(* Logix 5000 project; controller CHASKEY Emulate 5570 rev 30.12; software revision 30.00 *)

TASK MainTask (periodic, rate 3000 ms, priority 1, watchdog 5000 ms) : MainProgram

MODULES
   Local : Emulate 5570 (ICP 2, rev 30.12)
END_MODULES

VAR_GLOBAL   (* controller tags *)
   _SEC_P : BOOL;
   done : DINT;
   R_TRIG : FBD_ONESHOT;
   temp_var : DINT;
   test_array : DINT[20] := ([0] := 1, [1] := 2, [2] := 3, [3] := 4, [4] := 5, [5] := 6, [6] := 7, [7] := 8, [8] := 9, [9] := 10, [10] := 11, [11] := 12, [12] := 13, [13] := 14, [14] := 15, [15] := 16, [16] := 17, [17] := 18, [18] := 19, [19] := 20);
   TON : FBD_TIMER;
END_VAR

PROGRAM MainProgram   (* main routine MainRoutine *)
VAR
   Chaskey_128_i : DINT;
   Chaskey_a : DINT; {access None}
   Chaskey_AS_res : ALIAS FOR Chaskey_128_i;
   Chaskey_BNum : DINT; {access None}
   Chaskey_hi : DINT[4]; {access None}
   Chaskey_i : DINT; {access None}
   Chaskey_input_pi : DINT[4]; {access None}
   Chaskey_isPad : BOOL; {access None}
   Chaskey_j : DINT; {access None}
   Chaskey_key : DINT[4]; {access None}
   Chaskey_L : DINT[4]; {access None}
   Chaskey_LBLen : DINT; {access None}
   Chaskey_Message : DINT[256]; {access None}
   Chaskey_MsgBitLen : DINT; {access None}
   Chaskey_PadIndx1 : DINT; {access None}
   Chaskey_PadIndx2 : DINT; {access None}
   Chaskey_per_i : DINT; {access None}
   Chaskey_round : DINT;
   Chaskey_shift_input : DINT; {access None}
   Chaskey_shift_result : DINT; {access None}
   Chaskey_subkey1_i : DINT; {access None}
   Chaskey_subkey2_i : DINT; {access None}
   Chaskey_subkey_1 : DINT[8];
   Chaskey_subkey_2 : DINT[8]; {access None}
   Chaskey_tag : DINT[4]; {access None}
   Chaskey_Temp : DINT; {access None}
   PRG_Counter : DINT[2];
   PRG_i : DINT;
   PRG_j : DINT;
   PRG_Res_Len : DINT;
   PRG_Result : DINT[256];
   SCAN_CYCLE_TIME : DINT; {access None}
END_VAR

ROUTINE CHASKEY_128   (* structured text *)
   Chaskey_BNum:= Chaskey_MsgBitLen/128;
   
   
   if Chaskey_MsgBitLen mod 128 =0 then
   	Chaskey_isPad:=0;
   else
   	Chaskey_isPad:=1;
   	Chaskey_LBLen:= Chaskey_MsgBitLen - Chaskey_BNum*128;
   	Chaskey_PadIndx1 := (128 - Chaskey_LBLen)/32 + Chaskey_BNum/32;
   	Chaskey_PadIndx2 := ((128 - Chaskey_LBLen) mod 32) -1;
   	Chaskey_Message[Chaskey_PadIndx1]:= Chaskey_Message[Chaskey_PadIndx1]+ 10 ** Chaskey_PadIndx2;
   end_if;
   
   Chaskey_hi[3] := Chaskey_key[3];
   Chaskey_hi[2] := Chaskey_key[2] ;
   Chaskey_hi[1] := Chaskey_key[1] ;
   Chaskey_hi[0] := Chaskey_key[0] ;
   
   
   for Chaskey_i:=0 to Chaskey_BNum-1 do
   	Chaskey_128_i:=Chaskey_i*4;
   	Chaskey_input_pi[3] := Chaskey_hi[3] XOR Chaskey_Message[Chaskey_128_i+3] ;
   	Chaskey_input_pi[2] := Chaskey_hi[2] XOR Chaskey_Message[Chaskey_128_i+2] ;
   	Chaskey_input_pi[1] := Chaskey_hi[1] XOR Chaskey_Message[Chaskey_128_i+1] ;
   	Chaskey_input_pi[0] := Chaskey_hi[0] XOR Chaskey_Message[Chaskey_128_i+0] ;
   
   	JSR(CHASKEY_Permutation);
    	Chaskey_hi[3] := Chaskey_input_pi[3];
   	Chaskey_hi[2] := Chaskey_input_pi[2] ;
   	Chaskey_hi[1] := Chaskey_input_pi[1] ;
   	Chaskey_hi[0] := Chaskey_input_pi[0] ;
   
   	if Chaskey_i>=Chaskey_BNum-1 then
   		Exit;
   	end_if;
   
   end_for;
   
   if Chaskey_isPad then
   		//use K_2, run the final permutation
   	Chaskey_L[3] := Chaskey_subkey_2[3];
   	Chaskey_L[2] := Chaskey_subkey_2[2] ;
   	Chaskey_L[1] := Chaskey_subkey_2[1] ;
   	Chaskey_L[0] := Chaskey_subkey_2[0] ;
   else
   	Chaskey_L[3] := Chaskey_subkey_1[3];
   	Chaskey_L[2] := Chaskey_subkey_1[2] ;
   	Chaskey_L[1] := Chaskey_subkey_1[1] ;
   	Chaskey_L[0] := Chaskey_subkey_1[0] ;
   end_if;
   
   /*	if m_len > 128 then
   	chaskey_i:=chaskey_i+1;
   end_if;*/
   Chaskey_128_i:=Chaskey_i*4;
   Chaskey_input_pi[3] := Chaskey_hi[3] XOR Chaskey_Message[Chaskey_128_i+3] ;
   Chaskey_input_pi[2] := Chaskey_hi[2] XOR Chaskey_Message[Chaskey_128_i+2] ;
   Chaskey_input_pi[1] := Chaskey_hi[1] XOR Chaskey_Message[Chaskey_128_i+1] ;
   Chaskey_input_pi[0] := Chaskey_hi[0] XOR Chaskey_Message[Chaskey_128_i+0] ;
   
   Chaskey_input_pi[3] := Chaskey_input_pi[3] XOR Chaskey_L[3] ;
   Chaskey_input_pi[2] := Chaskey_input_pi[2] XOR Chaskey_L[2] ;
   Chaskey_input_pi[1] := Chaskey_input_pi[1] XOR Chaskey_L[1] ;
   Chaskey_input_pi[0] := Chaskey_input_pi[0] XOR Chaskey_L[0] ;
   
   JSR(CHASKEY_Permutation);
   
   Chaskey_input_pi[3] := Chaskey_input_pi[3] XOR Chaskey_L[3] ;
   Chaskey_input_pi[2] := Chaskey_input_pi[2] XOR Chaskey_L[2] ;
   Chaskey_input_pi[1] := Chaskey_input_pi[1] XOR Chaskey_L[1] ;
   Chaskey_input_pi[0] := Chaskey_input_pi[0] XOR Chaskey_L[0] ;
   
   //////////////////////////////////////////////
   
   
   Chaskey_tag[3] := Chaskey_input_pi[3];
   Chaskey_tag[2] := Chaskey_input_pi[2];
   Chaskey_tag[1] := Chaskey_input_pi[1];
   Chaskey_tag[0] := Chaskey_input_pi[0];
   
   JSR(CHASKEY_ClearKey);
   
END_ROUTINE

ROUTINE CHASKEY_ClearKey   (* structured text *)
   
   Chaskey_key[0]:= 0;
   Chaskey_key[1]:= 0;
   Chaskey_key[2]:= 0;
   Chaskey_key[3]:= 0;
   
   
   Chaskey_subkey_1[0]:= 0;
   Chaskey_subkey_1[1]:= 0;
   Chaskey_subkey_1[2]:= 0;
   Chaskey_subkey_1[3]:= 0;
   
   Chaskey_subkey_2[0]:= 0;
   Chaskey_subkey_2[1]:= 0;
   Chaskey_subkey_2[2]:= 0;
   Chaskey_subkey_2[3]:= 0;
   
END_ROUTINE

ROUTINE CHASKEY_Init   (* structured text *)
    //key[3].31 is the MSB of the key, while key[0].0 is the LSB of the key
   Chaskey_key[0]:=0;
   Chaskey_key[1]:=16#11;
   Chaskey_key[2]:=16#22;
   Chaskey_key[3]:=16#33;
   
   Chaskey_tag[0] := 0;
   Chaskey_tag[1] := 0;
   Chaskey_tag[2] := 0;
   Chaskey_tag[3] := 0;
   
   //Initialize subkey_1[] and subkey_2[]
   Chaskey_subkey_1[0] := 1715741319;
   Chaskey_subkey_1[1] := -288576888;
   Chaskey_subkey_1[2] := 2002070336;
   Chaskey_subkey_1[3] := -2245735;
   
   Chaskey_subkey_2[0] := -863484535;
   Chaskey_subkey_2[1] := -577153776;
   Chaskey_subkey_2[2] := -290822623;
   Chaskey_subkey_2[3] := -4491470;
   
   
   
END_ROUTINE

ROUTINE CHASKEY_Permutation   (* structured text *)
   
   for Chaskey_per_i:=0 to Chaskey_round by 1 do
   
   	//Chaskey_input_pi[0]:=Chaskey_input_pi[0] + Chaskey_input_pi[1];
   	Chaskey_input_pi[0]:= Chaskey_input_pi[0] + Chaskey_input_pi[1];
   	//Chaskey_input_pi[2]:=Chaskey_input_pi[2]+Chaskey_input_pi[3];
       Chaskey_input_pi[2]:= Chaskey_input_pi[2] + Chaskey_input_pi[3];
   
   	Chaskey_a:=Chaskey_input_pi[1];  //v1 <<< 5
   	Chaskey_Temp:=0;
   	//left shift Chaskey_b=5 bits
   	Chaskey_Temp.5:=Chaskey_a.0;
   	Chaskey_Temp.6:=Chaskey_a.1;
   	Chaskey_Temp.7:=Chaskey_a.2;
   	Chaskey_Temp.8:=Chaskey_a.3;
   	Chaskey_Temp.9:=Chaskey_a.4;
   	Chaskey_Temp.10:=Chaskey_a.5;
   	Chaskey_Temp.11:=Chaskey_a.6;
   	Chaskey_Temp.12:=Chaskey_a.7;
   	Chaskey_Temp.13:=Chaskey_a.8;
   	Chaskey_Temp.14:=Chaskey_a.9;
   	Chaskey_Temp.15:=Chaskey_a.10;
   	Chaskey_Temp.16:=Chaskey_a.11;
   	Chaskey_Temp.17:=Chaskey_a.12;
   	Chaskey_Temp.18:=Chaskey_a.13;
   	Chaskey_Temp.19:=Chaskey_a.14;
   	Chaskey_Temp.20:=Chaskey_a.15;
   	Chaskey_Temp.21:=Chaskey_a.16;
   	Chaskey_Temp.22:=Chaskey_a.17;
   	Chaskey_Temp.23:=Chaskey_a.18;
   	Chaskey_Temp.24:=Chaskey_a.19;
   	Chaskey_Temp.25:=Chaskey_a.20;
   	Chaskey_Temp.26:=Chaskey_a.21;
   	Chaskey_Temp.27:=Chaskey_a.22;
   	Chaskey_Temp.28:=Chaskey_a.23;
   	Chaskey_Temp.29:=Chaskey_a.24;
   	Chaskey_Temp.30:=Chaskey_a.25;
   	Chaskey_Temp.31:=Chaskey_a.26;
   	Chaskey_Temp.0:=Chaskey_a.27;
   	Chaskey_Temp.1:=Chaskey_a.28;
   	Chaskey_Temp.2:=Chaskey_a.29;
   	Chaskey_Temp.3:=Chaskey_a.30;
   	Chaskey_Temp.4:=Chaskey_a.31;
   
   	Chaskey_input_pi[1]:=Chaskey_Temp;
   	Chaskey_input_pi[1]:=Chaskey_input_pi[1] XOR Chaskey_input_pi[0];
   
   
   	Chaskey_a:=Chaskey_input_pi[0];  // <<< 16
   	Chaskey_Temp:=0;
   	//left shift Chaskey_b=16 bits
   	Chaskey_Temp.16:=Chaskey_a.0;
   	Chaskey_Temp.17:=Chaskey_a.1;
   	Chaskey_Temp.18:=Chaskey_a.2;
   	Chaskey_Temp.19:=Chaskey_a.3;
   	Chaskey_Temp.20:=Chaskey_a.4;
   	Chaskey_Temp.21:=Chaskey_a.5;
   	Chaskey_Temp.22:=Chaskey_a.5;
   	Chaskey_Temp.23:=Chaskey_a.7;
   	Chaskey_Temp.24:=Chaskey_a.8;
   	Chaskey_Temp.25:=Chaskey_a.9;
   	Chaskey_Temp.26:=Chaskey_a.10;
   	Chaskey_Temp.27:=Chaskey_a.11;
   	Chaskey_Temp.28:=Chaskey_a.12;
   	Chaskey_Temp.29:=Chaskey_a.13;
   	Chaskey_Temp.30:=Chaskey_a.14;
   	Chaskey_Temp.31:=Chaskey_a.15;
   	Chaskey_Temp.0:=Chaskey_a.16;
   	Chaskey_Temp.1:=Chaskey_a.17;
   	Chaskey_Temp.2:=Chaskey_a.18;
   	Chaskey_Temp.3:=Chaskey_a.19;
   	Chaskey_Temp.4:=Chaskey_a.20;
   	Chaskey_Temp.5:=Chaskey_a.21;
   	Chaskey_Temp.6:=Chaskey_a.22;
   	Chaskey_Temp.7:=Chaskey_a.23;
   	Chaskey_Temp.8:=Chaskey_a.24;
   	Chaskey_Temp.9:=Chaskey_a.25;
   	Chaskey_Temp.10:=Chaskey_a.26;
   	Chaskey_Temp.11:=Chaskey_a.27;
   	Chaskey_Temp.12:=Chaskey_a.28;
   	Chaskey_Temp.13:=Chaskey_a.29;
   	Chaskey_Temp.14:=Chaskey_a.30;
   	Chaskey_Temp.15:=Chaskey_a.31;
   
   	Chaskey_input_pi[0]:=Chaskey_Temp;
   
   
   	Chaskey_a:=Chaskey_input_pi[3];  // <<< 8
   	Chaskey_Temp:=0;
   	//left shift Chaskey_b=8 bits
   	Chaskey_Temp.8:=Chaskey_a.0;
   	Chaskey_Temp.9:=Chaskey_a.1;
   	Chaskey_Temp.10:=Chaskey_a.2;
   	Chaskey_Temp.11:=Chaskey_a.3;
   	Chaskey_Temp.12:=Chaskey_a.4;
   	Chaskey_Temp.13:=Chaskey_a.5;
   	Chaskey_Temp.14:=Chaskey_a.6;
   	Chaskey_Temp.15:=Chaskey_a.7;
   	Chaskey_Temp.16:=Chaskey_a.8;
   	Chaskey_Temp.17:=Chaskey_a.9;
   	Chaskey_Temp.18:=Chaskey_a.10;
   	Chaskey_Temp.19:=Chaskey_a.11;
   	Chaskey_Temp.20:=Chaskey_a.12;
   	Chaskey_Temp.21:=Chaskey_a.13;
   	Chaskey_Temp.22:=Chaskey_a.14;
   	Chaskey_Temp.23:=Chaskey_a.15;
   	Chaskey_Temp.24:=Chaskey_a.16;
   	Chaskey_Temp.25:=Chaskey_a.17;
   	Chaskey_Temp.26:=Chaskey_a.18;
   	Chaskey_Temp.27:=Chaskey_a.19;
   	Chaskey_Temp.28:=Chaskey_a.20;
   	Chaskey_Temp.29:=Chaskey_a.21;
   	Chaskey_Temp.30:=Chaskey_a.22;
   	Chaskey_Temp.31:=Chaskey_a.23;
   	Chaskey_Temp.0:=Chaskey_a.24;
   	Chaskey_Temp.1:=Chaskey_a.25;
   	Chaskey_Temp.2:=Chaskey_a.26;
   	Chaskey_Temp.3:=Chaskey_a.27;
   	Chaskey_Temp.4:=Chaskey_a.28;
   	Chaskey_Temp.5:=Chaskey_a.29;
   	Chaskey_Temp.6:=Chaskey_a.30;
   	Chaskey_Temp.7:=Chaskey_a.31;
   
   	Chaskey_input_pi[3]:=Chaskey_Temp;
   	Chaskey_input_pi[3]:=Chaskey_input_pi[3] XOR Chaskey_input_pi[2];
   
   
   	//Chaskey_input_pi[0]:=Chaskey_input_pi[0]+Chaskey_input_pi[3];
   	Chaskey_input_pi[0]:= Chaskey_input_pi[0] + Chaskey_input_pi[3];
   
   
   	Chaskey_a:=Chaskey_input_pi[3];  //<<< 13
   	Chaskey_Temp:=0;
   	//left shift Chaskey_b=13 bits
   	Chaskey_Temp.13:=Chaskey_a.0;
   	Chaskey_Temp.14:=Chaskey_a.1;
   	Chaskey_Temp.15:=Chaskey_a.2;
   	Chaskey_Temp.16:=Chaskey_a.3;
   	Chaskey_Temp.17:=Chaskey_a.4;
   	Chaskey_Temp.18:=Chaskey_a.5;
   	Chaskey_Temp.19:=Chaskey_a.6;
   	Chaskey_Temp.20:=Chaskey_a.7;
   	Chaskey_Temp.21:=Chaskey_a.8;
   	Chaskey_Temp.22:=Chaskey_a.9;
   	Chaskey_Temp.23:=Chaskey_a.10;
   	Chaskey_Temp.24:=Chaskey_a.11;
   	Chaskey_Temp.25:=Chaskey_a.12;
   	Chaskey_Temp.26:=Chaskey_a.13;
   	Chaskey_Temp.27:=Chaskey_a.14;
   	Chaskey_Temp.28:=Chaskey_a.15;
   	Chaskey_Temp.29:=Chaskey_a.16;
   	Chaskey_Temp.30:=Chaskey_a.17;
   	Chaskey_Temp.31:=Chaskey_a.18;
   	Chaskey_Temp.0:=Chaskey_a.19;
   	Chaskey_Temp.1:=Chaskey_a.20;
   	Chaskey_Temp.2:=Chaskey_a.21;
   	Chaskey_Temp.3:=Chaskey_a.22;
   	Chaskey_Temp.4:=Chaskey_a.23;
   	Chaskey_Temp.5:=Chaskey_a.24;
   	Chaskey_Temp.6:=Chaskey_a.25;
   	Chaskey_Temp.7:=Chaskey_a.26;
   	Chaskey_Temp.8:=Chaskey_a.27;
   	Chaskey_Temp.9:=Chaskey_a.28;
   	Chaskey_Temp.10:=Chaskey_a.29;
   	Chaskey_Temp.11:=Chaskey_a.30;
   
   	Chaskey_input_pi[3]:=Chaskey_Temp;
   	Chaskey_input_pi[3]:=Chaskey_input_pi[3] XOR Chaskey_input_pi[0];
   
   
   	//Chaskey_input_pi[2]:= Chaskey_input_pi[2] + Chaskey_input_pi[1];
   	Chaskey_input_pi[2]:=  Chaskey_input_pi[2] + Chaskey_input_pi[1];
   
   
   	Chaskey_a:=Chaskey_input_pi[1]; //<<< 7
   	Chaskey_Temp:=0;
   	//left shift Chaskey_b=7 bits
   	Chaskey_Temp.7:=Chaskey_a.0;
   	Chaskey_Temp.8:=Chaskey_a.1;
   	Chaskey_Temp.9:=Chaskey_a.2;
   	Chaskey_Temp.10:=Chaskey_a.3;
   	Chaskey_Temp.11:=Chaskey_a.4;
   	Chaskey_Temp.12:=Chaskey_a.5;
   	Chaskey_Temp.13:=Chaskey_a.6;
   	Chaskey_Temp.14:=Chaskey_a.7;
   	Chaskey_Temp.15:=Chaskey_a.8;
   	Chaskey_Temp.16:=Chaskey_a.9;
   	Chaskey_Temp.17:=Chaskey_a.10;
   	Chaskey_Temp.18:=Chaskey_a.11;
   	Chaskey_Temp.19:=Chaskey_a.12;
   	Chaskey_Temp.20:=Chaskey_a.13;
   	Chaskey_Temp.21:=Chaskey_a.14;
   	Chaskey_Temp.22:=Chaskey_a.15;
   	Chaskey_Temp.23:=Chaskey_a.16;
   	Chaskey_Temp.24:=Chaskey_a.17;
   	Chaskey_Temp.25:=Chaskey_a.18;
   	Chaskey_Temp.26:=Chaskey_a.19;
   	Chaskey_Temp.27:=Chaskey_a.20;
   	Chaskey_Temp.28:=Chaskey_a.21;
   	Chaskey_Temp.29:=Chaskey_a.22;
   	Chaskey_Temp.30:=Chaskey_a.23;
   	Chaskey_Temp.31:=Chaskey_a.24;
   	Chaskey_Temp.0:=Chaskey_a.25;
   	Chaskey_Temp.1:=Chaskey_a.26;
   	Chaskey_Temp.2:=Chaskey_a.27;
   	Chaskey_Temp.3:=Chaskey_a.28;
   	Chaskey_Temp.4:=Chaskey_a.29;
   	Chaskey_Temp.5:=Chaskey_a.30;
   	Chaskey_Temp.6:=Chaskey_a.31;
   
   	Chaskey_input_pi[1]:=Chaskey_Temp;
   	Chaskey_input_pi[1]:=Chaskey_input_pi[1] XOR Chaskey_input_pi[2];
   
   
   	Chaskey_a:=Chaskey_input_pi[2];   //<<< 16
   	Chaskey_Temp:=0;
   	//left shift Chaskey_b=16 bits
   	Chaskey_Temp.16:=Chaskey_a.0;
   	Chaskey_Temp.17:=Chaskey_a.1;
   	Chaskey_Temp.18:=Chaskey_a.2;
   	Chaskey_Temp.19:=Chaskey_a.3;
   	Chaskey_Temp.20:=Chaskey_a.4;
   	Chaskey_Temp.21:=Chaskey_a.5;
   	Chaskey_Temp.22:=Chaskey_a.5;
   	Chaskey_Temp.23:=Chaskey_a.7;
   	Chaskey_Temp.24:=Chaskey_a.8;
   	Chaskey_Temp.25:=Chaskey_a.9;
   	Chaskey_Temp.26:=Chaskey_a.10;
   	Chaskey_Temp.27:=Chaskey_a.11;
   	Chaskey_Temp.28:=Chaskey_a.12;
   	Chaskey_Temp.29:=Chaskey_a.13;
   	Chaskey_Temp.30:=Chaskey_a.14;
   	Chaskey_Temp.31:=Chaskey_a.15;
   	Chaskey_Temp.0:=Chaskey_a.16;
   	Chaskey_Temp.1:=Chaskey_a.17;
   	Chaskey_Temp.2:=Chaskey_a.18;
   	Chaskey_Temp.3:=Chaskey_a.19;
   	Chaskey_Temp.4:=Chaskey_a.20;
   	Chaskey_Temp.5:=Chaskey_a.21;
   	Chaskey_Temp.6:=Chaskey_a.22;
   	Chaskey_Temp.7:=Chaskey_a.23;
   	Chaskey_Temp.8:=Chaskey_a.24;
   	Chaskey_Temp.9:=Chaskey_a.25;
   	Chaskey_Temp.10:=Chaskey_a.26;
   	Chaskey_Temp.11:=Chaskey_a.27;
   	Chaskey_Temp.12:=Chaskey_a.28;
   	Chaskey_Temp.13:=Chaskey_a.29;
   	Chaskey_Temp.14:=Chaskey_a.30;
   	Chaskey_Temp.15:=Chaskey_a.31;
   
   	Chaskey_input_pi[2]:=Chaskey_Temp;
   end_for;
   
   
END_ROUTINE

ROUTINE MainRoutine   (* ladder *)
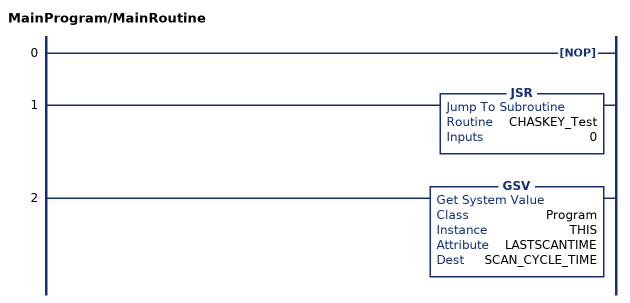
   0: NOP();
   1: JSR(CHASKEY_Test,0);
   2: GSV(Program,THIS,LASTSCANTIME,SCAN_CYCLE_TIME);
END_ROUTINE

ROUTINE PRG_PRF_CHASKEY   (* structured text *)
   JSR(PRG_PRF_Init);
   PRG_j:=0;
   For PRG_i:=0 to PRG_Res_Len by 1 do
   	Chaskey_Message[0]:=PRG_Counter[0]; //Upper bits of current plaintext
   	Chaskey_Message[1]:=PRG_Counter[1];  //Lower bits of current plaintext
   	Chaskey_Message[2]:=PRG_Counter[0]; //Upper bits of current plaintext
   	Chaskey_Message[3]:=PRG_Counter[1];  //Lower bits of current plaintext
   	JSR(CHASKEY_128);
   	PRG_Result[PRG_j]:=Chaskey_tag[0];
   	PRG_Result[PRG_j+1]:=Chaskey_tag[1];
   	PRG_Result[PRG_j+2]:=Chaskey_tag[2];
   	PRG_Result[PRG_j+3]:=Chaskey_tag[3];
   
   	PRG_j:=PRG_j+4;
   
   End_For;
   
   JSR(CHASKEY_ClearKey);
END_ROUTINE

ROUTINE PRG_PRF_CHASKEY_Test   (* structured text *)
   If S:FS Then
   
   	PRG_Counter[0]:=5;
   	PRG_Counter[1]:=1;
   
   
   End_if;
   
   
   JSR(PRG_PRF_CHASKEY);
   
   
END_ROUTINE

ROUTINE PRG_PRF_Init   (* structured text *)
   //initialize version
   
   
   Chaskey_round:=11;
   PRG_j:=0;
   PRG_Res_Len :=  (PRG_Counter[0] AND 16#0000ffff)-1;
   
   JSR(CHASKEY_Init);
END_ROUTINE
END_PROGRAM
